// Mitsubishi GX Works2 project: qr_robot_sort   PLC: Q03UDV

PROGRAM MAIN
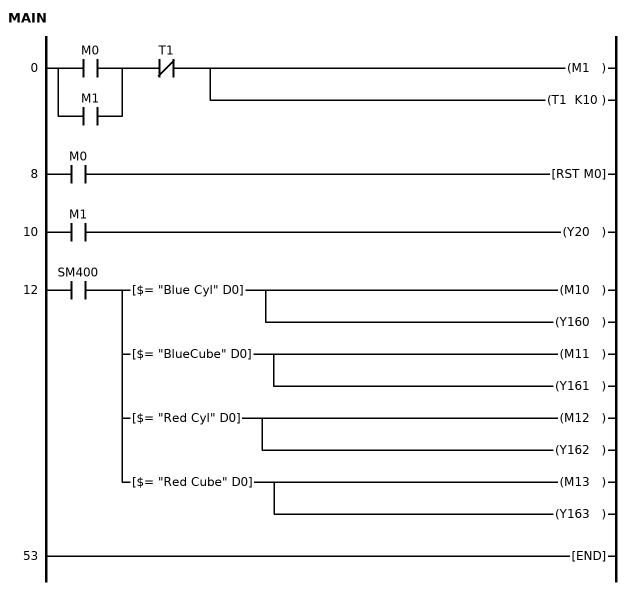
0     LD      M0
      OR      M1
      ANI     T1
      OUT     M1
      OUT     T1 K10
8     LD      M0
      RST     M0
10    LD      M1
      OUT     Y20
12    LD      SM400
      MPS
      AND$=   "Blue Cyl" D0
      OUT     M10
      OUT     Y160
      MRD
      AND$=   "BlueCube" D0
      OUT     M11
      OUT     Y161
      MRD
      AND$=   "Red Cyl" D0
      OUT     M12
      OUT     Y162
      MPP
      AND$=   "Red Cube" D0
      OUT     M13
      OUT     Y163
53    END
END_PROGRAM
